{attribute 'TcGenerated'}
{attribute 'no-analysis'}
{attribute 'linkalways'}
// This function has been automatically generated from the project information.
VAR_GLOBAL CONSTANT
    {attribute 'const_non_replaced'}
    stLibVersion_lcls_twincat_motion : ST_LibVersion := (iMajor := 0, iMinor := 0, iBuild := 0, iRevision := 0, nFlags := 0, sVersion := '0.0.0');
END_VAR

(* stored: Version 1.1.0.1
   GVL Global_Version: Id {e584f020-617f-4164-a737-6e483df3aa38} *)
